(* CODESYS project trafficLight.project

Project tree, tasks and I/O mapping:
  Device : CODESYS Control Win V3, 3S - Smart Software Solutions GmbH, order no. 305021, version 3.5.10.30
    application Application
      libraries: Standard, * (System)
      task MainTask (cyclic, interval t#20ms, priority 1) calls PLC_PRG
      task VISU_TASK (cyclic, interval 100 ms, priority 31) calls VisuElems.Visu_Prg
      program PLC_PRG [LD]
      safety/
        function block Emergency [LD]
        function block Anomalies [LD]
      visualisation Visualization
      fsm/
        function block TrafficLight [ST]
        function block TrafficLightBlinkingYellow [LD]
      cycle/
        function block Cycle [LD]
      output/
        function block UpdateOutput [LD]
  text list GlobalTextList
*)

// Device/Application/PLC_PRG
PROGRAM PLC_PRG
VAR
	// input
	btn_emergency AT %IX0.0 : BOOL := FALSE;
	btn_reset_anomalies AT %IX0.1 : BOOL := FALSE;
	aux AT %IX0.2 : BOOL := FALSE;
	
	switch_man_auto AT %IX1.0 : BOOL;
	btn_start_cycle AT %IX1.1 : BOOL;
	btn_user_request AT %IX1.2 : BOOL;
	light_sensor AT %IX1.3 : BOOL;
	
	tl_green_man AT %IX2.0 : BOOL := FALSE;
	tl_yellow_man AT %IX2.1 : BOOL := FALSE;
	tl_red_man AT %IX2.2 : BOOL := FALSE;

	// output
	tl_green AT %QX0.0 : BOOL := FALSE;
	tl_yellow AT %QX0.1 : BOOL := FALSE;
	tl_red AT %QX0.2 : BOOL := FALSE;
	
	// merker
	// var
	in_anomaly : BOOL;
	in_emergency : BOOL;
	man_auto : BOOL;
	tl_green_app : BOOL := FALSE;
	tl_yellow_app : BOOL := FALSE;
	tl_red_app : BOOL := FALSE;
	tlby_yellow_app : BOOL := false;
	
	anomalies : Anomalies;
	emergency : Emergency;
	cycle : Cycle;
	trafficLight: TrafficLight;
	trafficLightBlinkingYellow : TrafficLightBlinkingYellow;
	updateOutput : UpdateOutput;
	
END_VAR

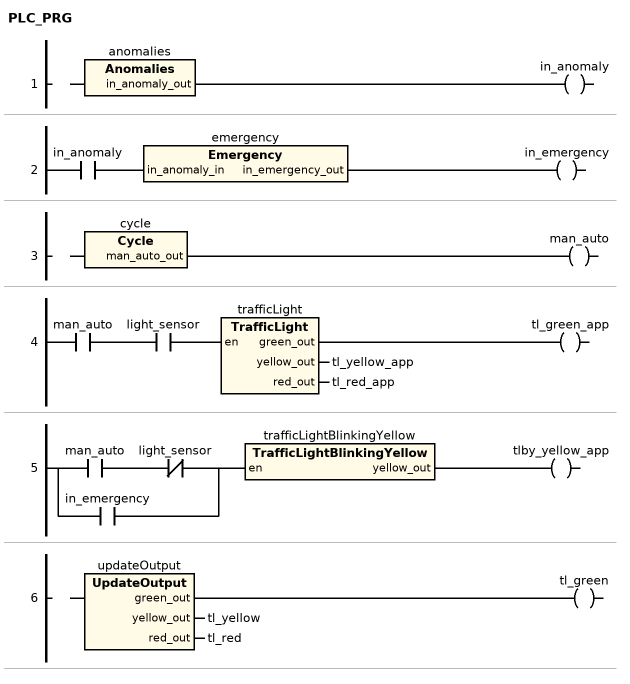
// NETWORK 1
anomalies();
in_anomaly := anomalies.in_anomaly_out;

// NETWORK 2
emergency(in_anomaly_in := in_anomaly);
in_emergency := emergency.in_emergency_out;

// NETWORK 3
cycle();
man_auto := cycle.man_auto_out;

// NETWORK 4
trafficLight(en := man_auto AND light_sensor, yellow_out => tl_yellow_app, red_out => tl_red_app);
tl_green_app := trafficLight.green_out;

// NETWORK 5
trafficLightBlinkingYellow(en := man_auto AND NOT light_sensor OR in_emergency);
tlby_yellow_app := trafficLightBlinkingYellow.yellow_out;

// NETWORK 6
updateOutput(yellow_out => tl_yellow, red_out => tl_red);
tl_green := updateOutput.green_out;

END_PROGRAM

// Device/Application/safety/Anomalies
FUNCTION_BLOCK Anomalies
VAR_INPUT
END_VAR
VAR_OUTPUT
	in_anomaly_out : BOOL;
END_VAR
VAR
	in_anomaly AT %MX0.1 : BOOL := FALSE;
	emergency_anomaly AT %MX1.0 : BOOL := FALSE;
	aux_anomaly AT %MX1.1 : BOOL := FALSE;
	other_anomaly_anomaly AT %MX1.1 : BOOL := FALSE;
	other_anomaly AT %MX2.1 : BOOL := FALSE;
END_VAR

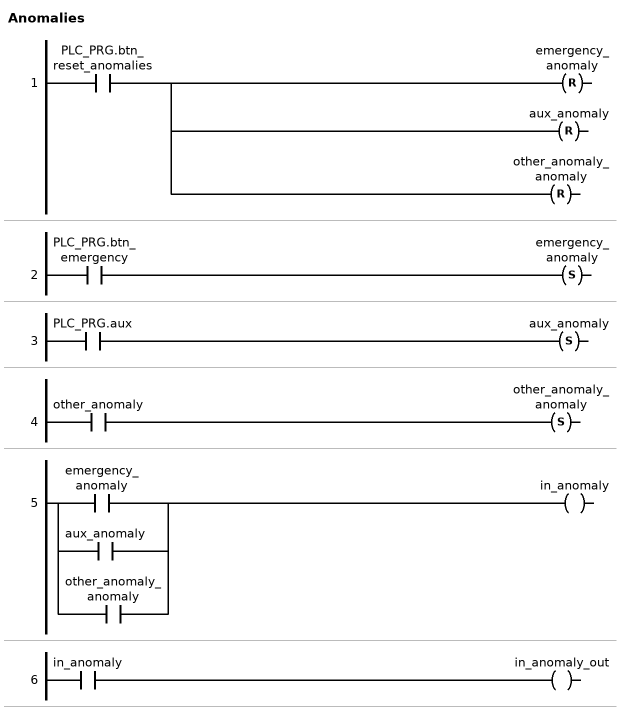
// NETWORK 1
emergency_anomaly R= PLC_PRG.btn_reset_anomalies;
aux_anomaly R= PLC_PRG.btn_reset_anomalies;
other_anomaly_anomaly R= PLC_PRG.btn_reset_anomalies;

// NETWORK 2
emergency_anomaly S= PLC_PRG.btn_emergency;

// NETWORK 3
aux_anomaly S= PLC_PRG.aux;

// NETWORK 4
other_anomaly_anomaly S= other_anomaly;

// NETWORK 5
in_anomaly := emergency_anomaly OR aux_anomaly OR other_anomaly_anomaly;

// NETWORK 6
in_anomaly_out := in_anomaly;

END_FUNCTION_BLOCK

// Device/Application/safety/Emergency
FUNCTION_BLOCK Emergency
VAR_INPUT
	in_anomaly_in : BOOL;
END_VAR
VAR_OUTPUT
	in_emergency_out : BOOL;
END_VAR
VAR
	in_emergency AT %MX0.0 : BOOL := FALSE;
END_VAR

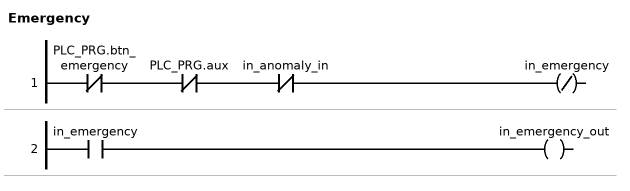
// NETWORK 1
in_emergency := NOT (NOT PLC_PRG.btn_emergency AND NOT PLC_PRG.aux AND NOT in_anomaly_in);

// NETWORK 2
in_emergency_out := in_emergency;

END_FUNCTION_BLOCK

// Device/Application/cycle/Cycle
FUNCTION_BLOCK Cycle
VAR_INPUT
END_VAR
VAR_OUTPUT
	man_auto_out : BOOL;
END_VAR
VAR
	man_auto AT %MX3.0 : BOOL := FALSE;
END_VAR

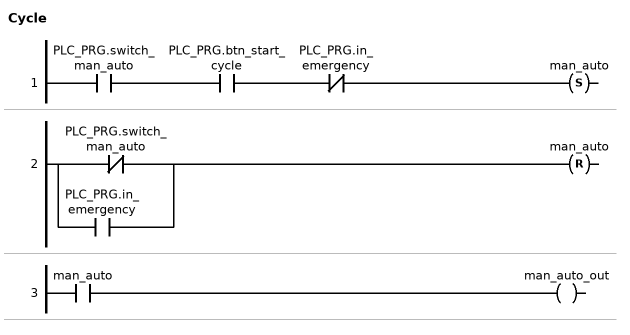
// NETWORK 1
man_auto S= PLC_PRG.switch_man_auto AND PLC_PRG.btn_start_cycle AND NOT PLC_PRG.in_emergency;

// NETWORK 2
man_auto R= NOT PLC_PRG.switch_man_auto OR PLC_PRG.in_emergency;

// NETWORK 3
man_auto_out := man_auto;

END_FUNCTION_BLOCK

// Device/Application/fsm/TrafficLight
FUNCTION_BLOCK TrafficLight
VAR_INPUT
	en : BOOL;
END_VAR
VAR_OUTPUT
	green_out : BOOL;
	yellow_out : BOOL;
	red_out : BOOL;

END_VAR

VAR
	state : INT := 0;
	ton_green : TON;
	ton_yellow : TON;
	ton_red : TON;
END_VAR

IF NOT en THEN
	state := 0;
	green_out := FALSE;
	yellow_out := FALSE;
	red_out := FALSE;
	ton_green(IN := FALSE, PT := T#1S);
	ton_yellow(IN := FALSE, PT := T#1S);
	ton_red(IN := FALSE, PT := T#1S);
	RETURN;
END_IF

CASE(state) OF
	0:
		state := 1;
	1:
		ton_green(IN := state=1, PT := T#5S);
		IF ton_green.q THEN
			state := 2;
			ton_green(IN := FALSE, PT := T#1S);
		END_IF
	2:
		ton_yellow(IN := state=2, PT := T#1S);
		IF ton_yellow.q THEN
			state := 3;
			ton_yellow(IN := FALSE, PT := T#1S);
		END_IF
	3:
		ton_red(IN := state=3, PT := T#3S);
		IF ton_red.q THEN
			state := 1;
			ton_red(IN := FALSE, PT := T#1S);
		END_IF
ELSE
	state := 0;
END_CASE

green_out := (state = 1);
yellow_out := (state = 2);
red_out := (state = 3);

END_FUNCTION_BLOCK

// Device/Application/fsm/TrafficLightBlinkingYellow
FUNCTION_BLOCK TrafficLightBlinkingYellow
VAR_INPUT
	en : BOOL;
END_VAR
VAR_OUTPUT
	yellow_out : BOOL;

END_VAR

VAR
	state : INT := 0;
	ton_yellow_on : TON;
	ton_yellow_off : TON;
END_VAR
VAR // added by the converter: edge detectors and wires of the graphical bodies
    _w1 : BOOL;
END_VAR

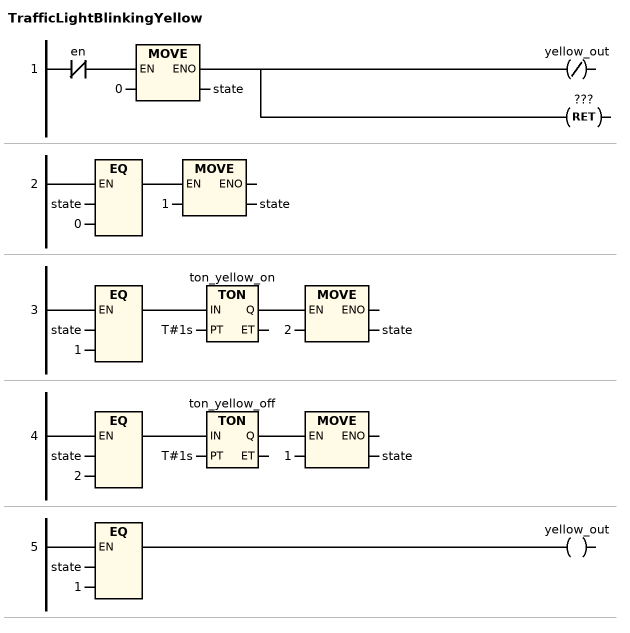
// NETWORK 1
_w1 := NOT en;
IF _w1 THEN state := 0; END_IF
yellow_out := NOT _w1;
IF _w1 THEN RETURN; END_IF

// NETWORK 2
IF state = 0 THEN state := 1; END_IF

// NETWORK 3
ton_yellow_on(IN := state = 1, PT := T#1s); // TON
IF ton_yellow_on.Q THEN state := 2; END_IF

// NETWORK 4
ton_yellow_off(IN := state = 2, PT := T#1s); // TON
IF ton_yellow_off.Q THEN state := 1; END_IF

// NETWORK 5
yellow_out := state = 1;

END_FUNCTION_BLOCK

// Device/Application/output/UpdateOutput
FUNCTION_BLOCK UpdateOutput
VAR_INPUT
END_VAR
VAR_OUTPUT
	green_out : BOOL;
	yellow_out : BOOL;
	red_out : BOOL;
END_VAR
VAR
END_VAR

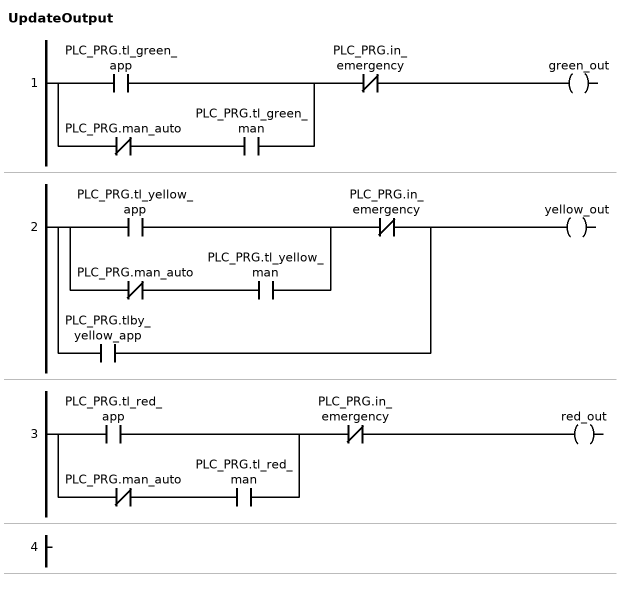
// NETWORK 1
green_out := (PLC_PRG.tl_green_app OR NOT PLC_PRG.man_auto AND PLC_PRG.tl_green_man) AND NOT PLC_PRG.in_emergency;

// NETWORK 2
yellow_out := (PLC_PRG.tl_yellow_app OR NOT PLC_PRG.man_auto AND PLC_PRG.tl_yellow_man) AND NOT PLC_PRG.in_emergency OR PLC_PRG.tlby_yellow_app;

// NETWORK 3
red_out := (PLC_PRG.tl_red_app OR NOT PLC_PRG.man_auto AND PLC_PRG.tl_red_man) AND NOT PLC_PRG.in_emergency;

// NETWORK 4

END_FUNCTION_BLOCK

// Device/Application/Visualization
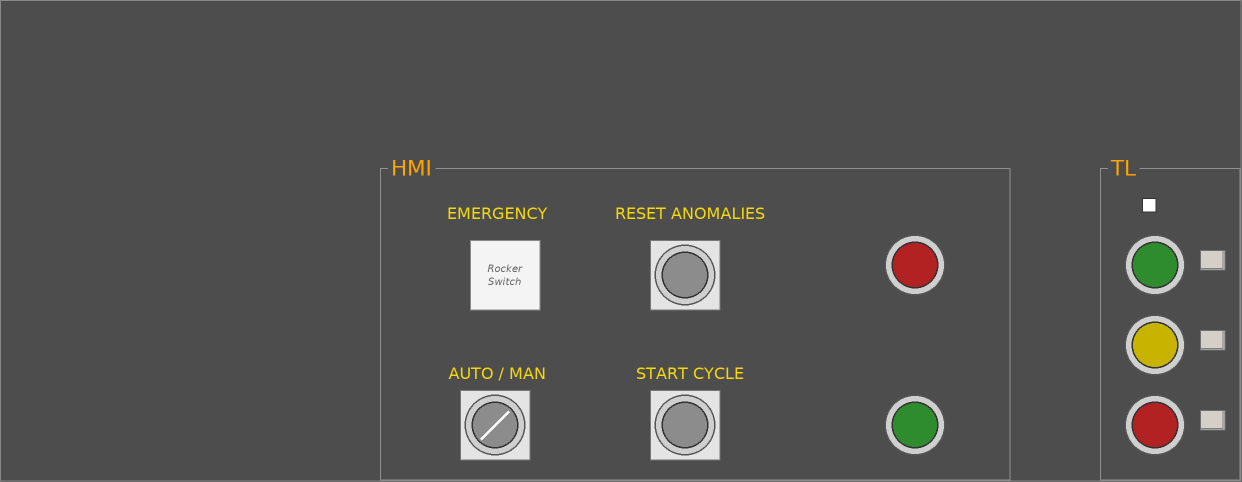
VISUALIZATION Visualization  // 1242x482
    Group (380,160 630x320)
        Lamp1 (500,70 70x70), variable: PLC_PRG.in_emergency, style: Lamp-Lamp1-Red
        PushSwitch (270,80 70x70), variable: PLC_PRG.btn_reset_anomalies, behaviour: TOGGLE, style: Switch-PushSwitch-Gray
        RockerSwitch (90,80 70x70), variable: PLC_PRG.btn_emergency, behaviour: TOGGLE, style: Switch-RockerSwitch-Gray
        PushSwitch (270,230 70x70), variable: PLC_PRG.btn_start_cycle, behaviour: TOGGLE, style: Switch-PushSwitch-Gray
        Lamp1 (500,230 70x70), variable: PLC_PRG.man_auto, style: Lamp-Lamp1-Green
        RotarySwitch (80,230 70x70), variable: PLC_PRG.switch_man_auto, behaviour: TOGGLE, style: Switch-RotarySwitch-Gray
        Label (60,40 115x27), "EMERGENCY"
        Label (210,40 200x27), "RESET ANOMALIES"
        Label (60,200 115x27), "AUTO / MAN"
        Label (240,200 140x27), "START CYCLE"
        GroupBox (0,0 630x320), "HMI"
    Group (1100,160 140x320)
        Lamp1 (20,230 70x70), variable: PLC_PRG.tl_red, style: Lamp-Lamp1-Red
        Lamp1 (20,150 70x70), variable: PLC_PRG.tl_yellow, style: Lamp-Lamp1-Yellow
        Lamp1 (20,70 70x70), variable: PLC_PRG.tl_green, style: Lamp-Lamp1-Green
        Checkbox (40,30 30x30), variable: PLC_PRG.light_sensor
        Button (100,90 25x20)
            tap PLC_PRG.tl_green_man
        Button (100,170 25x20)
            tap PLC_PRG.tl_yellow_man
        Button (100,250 25x20)
            tap PLC_PRG.tl_red_man
        GroupBox (0,0 140x320), "TL"
END_VISUALIZATION
